{attribute 'qualified_only'}
VAR_GLOBAL CONSTANT
	nEvents:						INT:= 49;		// Maximum of Events displayed in each Module
	tTimeout:						TIME:= T#5S;	// Default timeout for component pending states
END_VAR

(* stored: Version 1.1.0.1
   GVL Parameters: Id {a8306c1a-027b-005a-3454-c243d788d55f}, ParameterList True *)
